{attribute 'linkalways'} 
{attribute 'no_explicit_call' := 'This FB is a CLASS and must be accessed using methods or properties'}
{attribute 'enable_dynamic_creation'}
FUNCTION_BLOCK InputPort EXTENDS Disposable IMPLEMENTS I_InputPort
VAR
	_name : T_MAXSTRING;
	_data : I_Datatype;
	_connectedTo : I_OutputPort;
	parent : I_HaveInputPorts;
	eventEmitter : EventEmitter;
END_VAR

METHOD PUBLIC Accept
VAR_INPUT
	Visitor : I_InputPortVisitor;
END_VAR
Visitor.VisitInputPort(this^);
END_METHOD

PROPERTY PUBLIC Connected : BOOL
GET
Connected := _connectedTo <> 0;
END_GET
END_PROPERTY

METHOD PUBLIC ConnectTo
VAR_INPUT
	OutputPort : I_OutputPort;
END_VAR
_connectedTo := OutputPort;
_connectedTo.OnEvent('OnOutputPortChanged', THIS^);
END_METHOD

PROPERTY PUBLIC Data : I_Datatype
GET
Data := _data;
END_GET
END_PROPERTY

METHOD PUBLIC Disconnect
IF NOT Connected THEN
	RETURN;
END_IF

_connectedTo.OffEvent('OnOutputPortChanged', THIS^);
_connectedTo := 0;
END_METHOD

METHOD PROTECTED EmitOnInputPortChanged
VAR_INPUT
	PortChanged : I_InputPort;
END_VAR
VAR
	pInputPortChangeEvent : POINTER TO InputPortChangedEvent;
END_VAR
pInputPortChangeEvent := __NEW(InputPortChangedEvent(TargetInputPort := PortChanged));
eventEmitter.Emit('OnInputPortChanged',pInputPortChangeEvent^);
pInputPortChangeEvent^.Dispose();
END_METHOD

METHOD FB_init : BOOL
VAR_INPUT
	bInitRetains : BOOL; // if TRUE, the retain variables are initialized (warm start / cold start)
	bInCopyCode : BOOL;  // if TRUE, the instance afterwards gets moved into the copy code (online change)
	Name : T_MAXSTRING;
	Data : I_Datatype;
	Parent : I_HaveInputPorts;
END_VAR
_name := Name;
_data := Data;
RegisterWithParent(Parent);
END_METHOD

METHOD PUBLIC HandleEvent
VAR_INPUT
	Event : I_Event;
END_VAR
VAR
	outputPortChangedEvent : I_OutputPortChangedEvent;
END_VAR
IF __QUERYINTERFACE(Event, outputPortChangedEvent) THEN
	HandleOutputPortChangedEvent(outputPortChangedEvent.TargetOutputPort);
END_IF
END_METHOD

METHOD PROTECTED HandleOutputPortChangedEvent
VAR_INPUT
	Source : I_OutputPort;
END_VAR
EmitOnInputPortChanged(THIS^);
END_METHOD

PROPERTY PUBLIC Name : T_MAXSTRING
GET
Name := _name;
END_GET
END_PROPERTY

METHOD PUBLIC OffEvent
VAR_INPUT
	EventName : T_MaxString;
	EventHandler : I_EventHandler;
END_VAR
eventEmitter.OffEvent(EventName, EventHandler);
END_METHOD

METHOD PUBLIC OnceEvent
VAR_INPUT
	EventName : T_MaxString;
	EventHandler : I_EventHandler;
END_VAR
eventEmitter.OnceEvent(EventName, EventHandler);
END_METHOD

METHOD PUBLIC OnEvent
VAR_INPUT
	EventName : T_MaxString;
	EventHandler : I_EventHandler;
END_VAR
eventEmitter.OnEvent(EventName, EventHandler);
END_METHOD

METHOD PUBLIC RegisterWithParent
VAR_INPUT
	Parent : I_HaveInputPorts;
END_VAR
IF Parent = 0 THEN
	RETURN;
END_IF

THIS^.parent := Parent;
Parent.AddInputPort(THIS^);
END_METHOD

METHOD PUBLIC SerializeWith
VAR_INPUT
	Serializer : I_Serializer;
END_VAR
VAR 
	isConnected : BOOL := Connected;
END_VAR
Serializer.StartObject();
Serializer.AddKeyString('name',_name);
Serializer.AddKeyBool('connected',isConnected);
Serializer.Addkey('datatype');
_data.SerializeTypeWith(Serializer);
Serializer.AddkeyObject('value',_data);
Serializer.EndObject();
END_METHOD

END_FUNCTION_BLOCK

(* stored: Version 1.1.0.1, ProductVersion 3.1.4024.12
   POU InputPort: Id {8a76cd64-8399-006f-0213-1bb5b2341bca}, SpecialFunc None
   Folder Constructor: Id {c02273f4-e8fc-0d09-3c19-79f73fa57a1b}
   Folder Protected: Id {1f1fa75f-3537-0229-2498-8638fd4c140f}
   Method Accept: Id {1625d170-79e2-014d-2c2b-8ace06c47aa1}
   Property Connected: Id {0eeca197-140f-0917-0914-20aa772b83ae}
   Get Get: Id {7caf9676-d732-0ed2-375f-00350fceb01e}
   Method ConnectTo: Id {cf2a22c3-c119-0919-3767-3381d146e55b}
   Property Data: Id {f697d0c9-35bd-003b-2eed-d1db3a1aaa7d}
   Get Get: Id {9027c130-d714-0b66-2e0c-fed40c3b84cf}
   Method Disconnect: Id {2d2d97fa-faba-033e-23df-3b334614454b}
   Method EmitOnInputPortChanged: Id {7ac9cdfd-9dc5-4ff8-8987-c18d9fe1fa6d}
   Method FB_init: Id {85cb6971-3869-03dd-0362-0b78635177f7}
   Method HandleEvent: Id {a301251b-128e-042e-2c82-4ee90daa8459}
   Method HandleOutputPortChangedEvent: Id {9bdbd293-4e3d-0e2f-0079-1e62c2ac0372}
   Property Name: Id {bed621d8-5fb5-029d-2ec1-72a1805573da}
   Get Get: Id {81e0229a-69c1-0712-0a6c-c9c3a3d10c8f}
   Method OffEvent: Id {8831601f-10ed-0308-0255-7aeb488c0bb1}
   Method OnceEvent: Id {02751623-dd18-0013-0361-602d9e5793b3}
   Method OnEvent: Id {6400660c-9990-0d44-03fa-8885dfec75cf}
   Method RegisterWithParent: Id {99f5fd26-21c8-4b31-8e93-5757e5345969}
   Method SerializeWith: Id {baf1e5a1-8726-45d4-a3c3-4b5a88746bac} *)
